PROGRAM PRG_CODE_GetItemAIManual
VAR
	fbCase_DuplicatCheck		: FB_CASE_DuplicatCheck;
	
	(* Init function/method declarations*)
	rTrigDataInit		: R_TRIG;
	bDataInit			: BOOL;
	iOuter				: INT;
	iPack				: INT;
	sPackNum			: STRING;
	sOuterNum			: STRING;
	sPackCode			: STRING;
	
	(* Inputs *)
	bExecute							: BOOL;
	
	(* In/Out *)
	stProductInstruction				: ST_PCM_Status;
	stOuterBarcodeDuplicate				: ST_RejectItems;
	stOuterDuplicatedPackCodesFound		: ST_RejectItems;
	stCaseRejectReasons					: ST_RejectReasonsForCase;
	stRejectReasonForOuters				: ST_RejectReasonsForOuter;	
	stRejectReasonForPacks				: ST_RejectReasonsForPack;	
	
	stCACData 							: ST_CAC_Data;
	
	(* Outputs *)	
	bDone 					: BOOL;
	bBusy					: BOOL;

	bCACValid				: BOOL;
	sRejectCode				: T_MaxString;
	bIsDuplicateOuters		: BOOL;
	bIsDuplicatePacks		: BOOL;
	bReadyToValidate		: BOOL;
	
	stUpdateCACData 		: ST_CAC_Data;
	
	
END_VAR

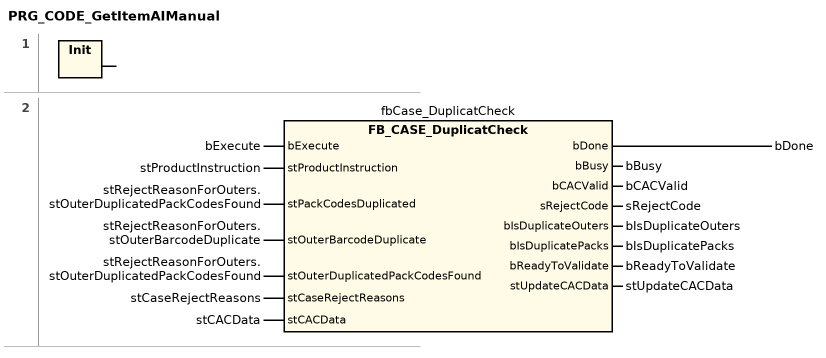
// NETWORK 1
Init();

// NETWORK 2
fbCase_DuplicatCheck(
    bExecute := bExecute,
    stProductInstruction := stProductInstruction,
    stPackCodesDuplicated := stRejectReasonForOuters.stOuterDuplicatedPackCodesFound,
    stOuterBarcodeDuplicate := stRejectReasonForOuters.stOuterBarcodeDuplicate,
    stOuterDuplicatedPackCodesFound := stRejectReasonForOuters.stOuterDuplicatedPackCodesFound,
    stCaseRejectReasons := stCaseRejectReasons,
    stCACData := stCACData,
    bBusy => bBusy,
    bCACValid => bCACValid,
    sRejectCode => sRejectCode,
    bIsDuplicateOuters => bIsDuplicateOuters,
    bIsDuplicatePacks => bIsDuplicatePacks,
    bReadyToValidate => bReadyToValidate,
    stUpdateCACData => stUpdateCACData); // FB_CASE_DuplicatCheck
bDone := fbCase_DuplicatCheck.bDone;

ACTION Init:

rTrigDataInit(CLK := bDataInit);

IF rTrigDataInit.Q THEN
	
stProductInstruction.nOutersPerCase		:= 50;
stProductInstruction.nPacksPerOuter 	:= 10;

	FOR iOuter := 1 TO stProductInstruction.nOutersPerCase DO
		(* Outer number z zerami *)
		sOuterNum := F_StringAddPrefix(INT_TO_STRING(iOuter),2,'0');
		
		(* Write Outers barcodes *)
		stCACData.Outer[iOuter].Barcode    := CONCAT('OUTER', sOuterNum);
		stCACData.Outer[iOuter].OuterCodeStatus := 5;
		
		FOR iPack := 1 TO stProductInstruction.nPacksPerOuter DO
			(* Pack number dwucyfrowy z zerami *)
			sPackNum := F_StringAddPrefix(INT_TO_STRING(iPack),2,'0');			
			(* Sklej pack code *)
			sPackCode := CONCAT(CONCAT('PACK', sPackNum), CONCAT('OUTER', sOuterNum));
			
			(* Write Pack Barcodes *)
			stCACData.Outer[iOuter].PackCode[iPack]			:= sPackCode;
			stCACData.Outer[iOuter].PackCodeStatus[iPack]	:= 5;
			stCACData.Outer[iOuter].PackRejectID[iPack]		:= 0;
			
		END_FOR;
	END_FOR;	
	
END_IF
END_ACTION

END_PROGRAM

(* stored: Version 1.1.0.1
   POU PRG_CODE_GetItemAIManual: Id {dff04167-7d63-4e54-ae52-95120ff519c5}, SpecialFunc None
   Action Init: Id {82e374ac-3a1c-4ce3-97a1-fb1ecbadc4a3} *)
